# B&R Automation Studio project arm
Automation Studio 4.2.10.53 SP

## Configuration Config1

CPU X20CP1586, AutomationRuntime D4.26, Build 4.1.2, Vc V4.26.5

### Task classes (Cpu.sw)
```
Cyclic#2 (cycle 20000 us, tolerance 20000 us):
  Program <- Program.prg
VcDataObjects: Visu <- Visu.dob
Binaries: TCData, arconfig, asfw, OpcUaMap, ashwd, iomap, User, Role, sysconf
Libraries: runtime, robot, astime, asieccon
```

### Hardware
```
X20CP1586 : X20CP1586 v1.3.0.0
  Connector IF1:
    ActivateIna = 0
  Connector IF2:
    ActivateDevice = 1
    EthInterfaceRedundant = 0
    InaPort = 11160
    Vnc1
    VncVcObjectName1 = Visu
    VncKeyMappingFile1 = VC\PS2-Keyboard.dis
  Connector IF3:
    EplInterfaceRedundant = 0
    EplEthInterfaceRedundant = 0
  ConfigurationID = arm_Config1
  Simulation = 1
  TimerDeviceType = SWIOTIMER
  Cyclic1Duration = 10000
  Cyclic1Tolerance = 10000
  Cyclic2Duration = 20000
  Cyclic2Tolerance = 20000
  Cyclic3Duration = 50000
  Cyclic3Tolerance = 50000
  Cyclic4Duration = 100000
  Cyclic4Tolerance = 100000
  Cyclic5Duration = 200000
  Cyclic5Tolerance = 200000
  Cyclic6Duration = 500000
  Cyclic6Tolerance = 500000
  Cyclic7Duration = 1000000
  Cyclic7Tolerance = 1000000
  Cyclic8Duration = 10000
  Cyclic8Tolerance = 30000000
  ActivateOpcUa = 1
  OpcUa_Security_SoftwareCertificates = 
  OpcUa_Security_AdminRole = 
```

## Logical view

Binary libraries used (declarations not repeated): operator, runtime, astime, AsIecCon

### Package Logical/Libraries - Global libraries

### Library Logical/Libraries/robot (IEC)

#### Types.typ - Exported data types
```iecst
TYPE
	AnimState :
		(
		IDLE,
		ANIMATING,
		ANIMATION_END
		);
END_TYPE
```

#### Constants.var - Exported constants
```iecst
VAR CONSTANT
	ANIMATING : USINT := 1;
	ANIMATION_END : USINT := 2;
END_VAR
```

#### robot.fun - Exported functions and function blocks
```iecst
FUNCTION_BLOCK Q_PositionAnimator (*TODO: Add your comment here*) (*$GROUP=User,$CAT=User,$GROUPICON=User.png,$CATICON=User.png*)
	VAR_INPUT
		startPosition : REAL := 0.0;
		endPosition : REAL := 0.0;
		reverse : BOOL := FALSE;
		enabled : BOOL := FALSE;
		velocity : INT := 1;
	END_VAR
	VAR_OUTPUT
		status : AnimState := IDLE;
		position : REAL;
	END_VAR
END_FUNCTION_BLOCK
```

#### Q_PositionAnimator.ab
```automation-basic
(* TODO: Add your comment here *)
FUNCTION_BLOCK Q_PositionAnimator
	IF enabled = TRUE THEN
		IF status <> ANIMATING THEN
			IF reverse = FALSE THEN
				position = startPosition
			ELSE
				position = endPosition
			ENDIF
			status = ANIMATING
		ENDIF
		IF startPosition = endPosition THEN
			status = ANIMATION_END
		ELSE
			IF reverse = FALSE THEN
				IF (startPosition - endPosition) < 0 THEN
					position = position + velocity
					IF position = endPosition THEN
						status = ANIMATION_END
					ENDIF
				ELSE
					position = position - velocity
					IF position = endPosition THEN
						status = ANIMATION_END
					ENDIF
				ENDIF
			ELSE
				IF (startPosition - endPosition) > 0 THEN
					position = position + velocity
					IF position = startPosition THEN
						status = ANIMATION_END
					ENDIF
				ELSE
					position = position - velocity
					IF position = startPosition THEN
						status = ANIMATION_END
					ENDIF
				ENDIF
			ENDIF
		ENDIF
	ELSE
		status = ANIMATION_END
	ENDIF
END_FUNCTION_BLOCK
```

### Program Logical/Program (IEC)

#### Cyclic.ab - Cyclic code
```automation-basic
PROGRAM _CYCLIC
	IF Visu_applyBtn = TRUE THEN
		platformMinAngle = REAL(Visu_PlatformMinAngle)
		platformMaxAngle = REAL(Visu_PlatformMaxAngle)
		shoulderMinAngle = REAL(Visu_ShoulderMinAngle)
		shoulderMaxAngle = REAL(Visu_ShoulderMaxAngle)
		localTranslateXnew = REAL(Visu_RobotTranslateX)
		localTranslateYnew = REAL(Visu_RobotTranslateY)
		localTranslateZnew = REAL(Visu_RobotTranslateZ)
		Q_PositionAnimator_0.enabled = FALSE
		Q_PositionAnimator_0 FUB Q_PositionAnimator()
		animationStep = 0
		Visu_applyBtn = FALSE
	ENDIF
	Q_PositionAnimator_0.enabled = TRUE
	SELECT animationStep
		STATE Q0Rotation
			Q_PositionAnimator_0.startPosition = platformMinAngle
			Q_PositionAnimator_0.endPosition = platformMaxAngle
			Q_PositionAnimator_0 FUB Q_PositionAnimator()
			robotManipulator.Position[0] = Q_PositionAnimator_0.position
			WHEN Q_PositionAnimator_0.status = ANIMATION_END
				NEXT Q1Rotation
		STATE Q1Rotation
			Q_PositionAnimator_0.startPosition = shoulderMinAngle
			Q_PositionAnimator_0.endPosition = shoulderMaxAngle
			Q_PositionAnimator_0 FUB Q_PositionAnimator()
			robotManipulator.Position[1] = Q_PositionAnimator_0.position
			WHEN Q_PositionAnimator_0.status = ANIMATION_END
				Q_PositionAnimator_0.velocity = 10
				tempReverse = Q_PositionAnimator_0.reverse
				Q_PositionAnimator_0.reverse = FALSE
				NEXT QX
		STATE QX
			WHEN localTranslateXold = localTranslateXnew
				NEXT QY
			Q_PositionAnimator_0.startPosition = localTranslateXold
			Q_PositionAnimator_0.endPosition = localTranslateXnew
			Q_PositionAnimator_0 FUB Q_PositionAnimator()
			robotManipulator.RobotTranslateX = Q_PositionAnimator_0.position
			WHEN Q_PositionAnimator_0.status = ANIMATION_END
				localTranslateXold = localTranslateXnew
				NEXT QY
		STATE QY
			WHEN localTranslateYold = localTranslateYnew
				NEXT QZ
			Q_PositionAnimator_0.startPosition = localTranslateYold
			Q_PositionAnimator_0.endPosition = localTranslateYnew
			Q_PositionAnimator_0 FUB Q_PositionAnimator()
			robotManipulator.RobotTranslateY = Q_PositionAnimator_0.position
			WHEN Q_PositionAnimator_0.status = ANIMATION_END
				localTranslateYold = localTranslateYnew
				NEXT QZ
		STATE QZ
			WHEN localTranslateZold = localTranslateZnew
				Q_PositionAnimator_0.velocity = 1
				Q_PositionAnimator_0.reverse = tempReverse
				NEXT ReverseAnimation
			Q_PositionAnimator_0.startPosition = localTranslateZold
			Q_PositionAnimator_0.endPosition = localTranslateZnew
			Q_PositionAnimator_0 FUB Q_PositionAnimator()
			robotManipulator.RobotTranslateZ = Q_PositionAnimator_0.position
			WHEN Q_PositionAnimator_0.status = ANIMATION_END
				localTranslateZold = localTranslateZnew
				Q_PositionAnimator_0.velocity = 1
				Q_PositionAnimator_0.reverse = tempReverse
				NEXT ReverseAnimation
		STATE ReverseAnimation
			reverse = NOT reverse
			Q_PositionAnimator_0.reverse = reverse
			WHEN TRUE
				NEXT Q0Rotation
	ENDSELECT
END_PROGRAM
```

#### Init.ab - Init code
```automation-basic
PROGRAM _INIT

END_PROGRAM
```

#### Types.typ - Local data types
```iecst
TYPE
	RobotManipulator : 	STRUCT
		RobotTranslateX : REAL;
		Position : ARRAY[0..6]OF REAL;
		RobotTranslateY : REAL;
		RobotTranslateZ : REAL;
		RobotTCPC : REAL;
		RobotTCPB : REAL;
		RobotTCPA : REAL;
	END_STRUCT;
END_TYPE
```

#### Variables.var - Local variables
```iecst
VAR
	shoulderMinAngle : REAL := 0;
	shoulderMaxAngle : REAL := 0.0;
	robotManipulator : RobotManipulator;
	reverse : BOOL := FALSE;
END_VAR
VAR RETAIN
	Q_PositionAnimator_0 : Q_PositionAnimator;
END_VAR
VAR
	platformMinAngle : REAL := 0;
	oneBigTrigger : BOOL := FALSE;
	platformMaxAngle : REAL := 0;
	animationStep : INT;
	Visu_RobotTranslateZ : INT;
	Visu_RobotTranslateY : INT;
	Visu_PlatformMinAngle : INT;
	Visu_PlatformMaxAngle : INT;
	Visu_ShoulderMinAngle : INT;
	Visu_ShoulderMaxAngle : INT;
	Visu_applyBtn : BOOL := FALSE;
	Visu_RobotTranslateX : INT;
	localTranslateXnew : REAL;
	localTranslateYnew : REAL;
	localTranslateZnew : REAL;
	localTranslateXold : REAL := 0;
	localTranslateYold : REAL := 0;
	localTranslateZold : REAL := 0;
	tempReverse : BOOL;
END_VAR
```

- Visualisation Logical/Visu (not shown)

Listed in the project but not available here: Logical/Global.typ, Logical/Global.var, Logical/Program/Exit.ab
